GLOBALCONSTANTS DefaultPool_AIC_3P (* Global constants *)
  PACKAGE Uebungen::const::UT::AIC;
  VAR_GLOBAL CONSTANT
    ISO_DESIGNATOR_WIDTH : UINT := 80;
    ISO_DESIGNATOR_HEIGHT : UINT := 80;
    ISO_MASK_SIZE : UINT := 480;
    ISO_VERSION_LABEL : STRING;
    MASK_WIDTH : UINT := 480;
    MASK_HEIGHT : UINT := 480;
    WorkingSet : UINT := 0;
    Macro_M1 : UINT := 1;
    Macro_AIC_1 : UINT := 2;
    Macro_AIC_2 : UINT := 3;
    Macro_AIC_3 : UINT := 4;
    Macro_AIC_4 : UINT := 5;
    DataMask_M1 : UINT := 1000;
    DataMask_AIC1 : UINT := 1001;
    DataMask_AIC2 : UINT := 1002;
    DataMask_AIC3 : UINT := 1003;
    DataMask_AIC4 : UINT := 1004;
    Container_Q : UINT := 3000;
    SoftKeyMask_AIC : UINT := 4000;
    SoftKey_Ausgaenge : UINT := 5000;
    SoftKey_AIC1 : UINT := 5001;
    SoftKey_AIC2 : UINT := 5002;
    SoftKey_AIC3 : UINT := 5003;
    SoftKey_AIC4 : UINT := 5004;
    Button_Q01 : UINT := 6001;
    Button_Q02 : UINT := 6002;
    Button_Q03 : UINT := 6003;
    Button_Q04 : UINT := 6004;
    Button_Q05 : UINT := 6005;
    Button_Q06 : UINT := 6006;
    Button_Q07 : UINT := 6007;
    Button_Q08 : UINT := 6008;
    Button_Q09 : UINT := 6009;
    Button_Q10 : UINT := 6010;
    Button_Q11 : UINT := 6011;
    Button_Q12 : UINT := 6012;
    Button_AIC_I01_CO : UINT := 6013;
    Button_AIC_I01_CS : UINT := 6014;
    Button_AIC_I02_CO : UINT := 6015;
    Button_AIC_I02_CS : UINT := 6016;
    Button_AIC_I03_CO : UINT := 6017;
    Button_AIC_I03_CS : UINT := 6018;
    Button_AIC_I04_CO : UINT := 6019;
    Button_AIC_I04_CS : UINT := 6020;
    Button_AIC_I05_CO : UINT := 6021;
    Button_AIC_I05_CS : UINT := 6022;
    Button_AIC_I06_CO : UINT := 6023;
    Button_AIC_I06_CS : UINT := 6024;
    Button_AIC_I07_CO : UINT := 6025;
    Button_AIC_I07_CS : UINT := 6026;
    Button_AIC_I08_CO : UINT := 6027;
    Button_AIC_I08_CS : UINT := 6028;
    Button_AIC_I01_MID : UINT := 6029;
    Button_AIC_I02_MID : UINT := 6030;
    Button_AIC_I03_MID : UINT := 6031;
    Button_AIC_I04_MID : UINT := 6032;
    Button_AIC_I05_MID : UINT := 6033;
    Button_AIC_I06_MID : UINT := 6034;
    Button_AIC_I07_MID : UINT := 6035;
    Button_AIC_I08_MID : UINT := 6036;
    InputNumber_AIC_I01_ZERO : UINT := 9000;
    InputNumber_AIC_I01_SPAN : UINT := 9001;
    InputNumber_AIC_I02_ZERO : UINT := 9002;
    InputNumber_AIC_I02_SPAN : UINT := 9003;
    InputNumber_AIC_I03_ZERO : UINT := 9004;
    InputNumber_AIC_I03_SPAN : UINT := 9005;
    InputNumber_AIC_I04_ZERO : UINT := 9006;
    InputNumber_AIC_I04_SPAN : UINT := 9007;
    InputNumber_AIC_I05_ZERO : UINT := 9008;
    InputNumber_AIC_I05_SPAN : UINT := 9009;
    InputNumber_AIC_I06_ZERO : UINT := 9010;
    InputNumber_AIC_I06_SPAN : UINT := 9011;
    InputNumber_AIC_I07_ZERO : UINT := 9012;
    InputNumber_AIC_I07_SPAN : UINT := 9013;
    InputNumber_AIC_I08_ZERO : UINT := 9014;
    InputNumber_AIC_I08_SPAN : UINT := 9015;
    InputNumber_AIC_I01_MID : UINT := 9016;
    InputNumber_AIC_I02_MID : UINT := 9017;
    InputNumber_AIC_I03_MID : UINT := 9018;
    InputNumber_AIC_I04_MID : UINT := 9019;
    InputNumber_AIC_I05_MID : UINT := 9020;
    InputNumber_AIC_I06_MID : UINT := 9021;
    InputNumber_AIC_I07_MID : UINT := 9022;
    InputNumber_AIC_I08_MID : UINT := 9023;
    OutputString_WorkingSet_0 : UINT := 11000;
    Label_SoftKey_Ausgaenge : UINT := 11001;
    Label_SoftKey_AIC1 : UINT := 11002;
    Label_SoftKey_AIC2 : UINT := 11003;
    Label_SoftKey_AIC3 : UINT := 11004;
    Label_SoftKey_AIC4 : UINT := 11005;
    Label_AIC_I01 : UINT := 11006;
    Label_AIC_I02 : UINT := 11007;
    Label_AIC_I03 : UINT := 11008;
    Label_AIC_I04 : UINT := 11009;
    Label_AIC_I05 : UINT := 11010;
    Label_AIC_I06 : UINT := 11011;
    Label_AIC_I07 : UINT := 11012;
    Label_AIC_I08 : UINT := 11013;
    Caption_MIN : UINT := 11014;
    Caption_MAX : UINT := 11015;
    Caption_MID : UINT := 11016;
    OutputNumber_c1 : UINT := 12001;
    OutputNumber_c9 : UINT := 12009;
    OutputNumber_c10 : UINT := 12010;
    OutputNumber_c11 : UINT := 12011;
    OutputNumber_c12 : UINT := 12012;
    OutputNumber_c2 : UINT := 12013;
    OutputNumber_c3 : UINT := 12014;
    OutputNumber_c4 : UINT := 12015;
    OutputNumber_c5 : UINT := 12016;
    OutputNumber_c6 : UINT := 12017;
    OutputNumber_c7 : UINT := 12018;
    OutputNumber_c8 : UINT := 12019;
    OutputNumber_Tick : UINT := 12020;
    OutputNumber_AIC_I01_RAW : UINT := 12021;
    OutputNumber_AIC_I01_CAL : UINT := 12022;
    OutputNumber_AIC_I02_RAW : UINT := 12023;
    OutputNumber_AIC_I02_CAL : UINT := 12024;
    OutputNumber_AIC_I03_RAW : UINT := 12025;
    OutputNumber_AIC_I03_CAL : UINT := 12026;
    OutputNumber_AIC_I04_RAW : UINT := 12027;
    OutputNumber_AIC_I04_CAL : UINT := 12028;
    OutputNumber_AIC_I05_RAW : UINT := 12029;
    OutputNumber_AIC_I05_CAL : UINT := 12030;
    OutputNumber_AIC_I06_RAW : UINT := 12031;
    OutputNumber_AIC_I06_CAL : UINT := 12032;
    OutputNumber_AIC_I07_RAW : UINT := 12033;
    OutputNumber_AIC_I07_CAL : UINT := 12034;
    OutputNumber_AIC_I08_RAW : UINT := 12035;
    OutputNumber_AIC_I08_CAL : UINT := 12036;
    OutputNumber_AIC_I01_MINRAW : UINT := 12037;
    OutputNumber_AIC_I01_MIDRAW : UINT := 12038;
    OutputNumber_AIC_I01_MAXRAW : UINT := 12039;
    OutputNumber_AIC_I02_MINRAW : UINT := 12040;
    OutputNumber_AIC_I02_MIDRAW : UINT := 12041;
    OutputNumber_AIC_I02_MAXRAW : UINT := 12042;
    OutputNumber_AIC_I03_MINRAW : UINT := 12043;
    OutputNumber_AIC_I03_MIDRAW : UINT := 12044;
    OutputNumber_AIC_I03_MAXRAW : UINT := 12045;
    OutputNumber_AIC_I04_MINRAW : UINT := 12046;
    OutputNumber_AIC_I04_MIDRAW : UINT := 12047;
    OutputNumber_AIC_I04_MAXRAW : UINT := 12048;
    OutputNumber_AIC_I05_MINRAW : UINT := 12049;
    OutputNumber_AIC_I05_MIDRAW : UINT := 12050;
    OutputNumber_AIC_I05_MAXRAW : UINT := 12051;
    OutputNumber_AIC_I06_MINRAW : UINT := 12052;
    OutputNumber_AIC_I06_MIDRAW : UINT := 12053;
    OutputNumber_AIC_I06_MAXRAW : UINT := 12054;
    OutputNumber_AIC_I07_MINRAW : UINT := 12055;
    OutputNumber_AIC_I07_MIDRAW : UINT := 12056;
    OutputNumber_AIC_I07_MAXRAW : UINT := 12057;
    OutputNumber_AIC_I08_MINRAW : UINT := 12058;
    OutputNumber_AIC_I08_MIDRAW : UINT := 12059;
    OutputNumber_AIC_I08_MAXRAW : UINT := 12060;
    Bargraph_AIC_I01 : UINT := 18000;
    Bargraph_AIC_I02 : UINT := 18001;
    Bargraph_AIC_I03 : UINT := 18002;
    Bargraph_AIC_I04 : UINT := 18003;
    Bargraph_AIC_I05 : UINT := 18004;
    Bargraph_AIC_I06 : UINT := 18005;
    Bargraph_AIC_I07 : UINT := 18006;
    Bargraph_AIC_I08 : UINT := 18007;
    Logos_icon : UINT := 20500;
    NumberVariable_AIC_RAW_I01 : UINT := 21000;
    NumberVariable_AIC_RAW_I02 : UINT := 21001;
    NumberVariable_AIC_RAW_I03 : UINT := 21002;
    NumberVariable_AIC_RAW_I04 : UINT := 21003;
    NumberVariable_AIC_RAW_I05 : UINT := 21004;
    NumberVariable_AIC_RAW_I06 : UINT := 21005;
    NumberVariable_AIC_RAW_I07 : UINT := 21006;
    NumberVariable_AIC_RAW_I08 : UINT := 21007;
    NumberVariable_AIC_CAL_I01 : UINT := 21008;
    NumberVariable_AIC_CAL_I02 : UINT := 21009;
    NumberVariable_AIC_CAL_I03 : UINT := 21010;
    NumberVariable_AIC_CAL_I04 : UINT := 21011;
    NumberVariable_AIC_CAL_I05 : UINT := 21012;
    NumberVariable_AIC_CAL_I06 : UINT := 21013;
    NumberVariable_AIC_CAL_I07 : UINT := 21014;
    NumberVariable_AIC_CAL_I08 : UINT := 21015;
    NumberVariable_AIC_I01_ZERO : UINT := 21016;
    NumberVariable_AIC_I01_SPAN : UINT := 21017;
    NumberVariable_AIC_I02_ZERO : UINT := 21018;
    NumberVariable_AIC_I02_SPAN : UINT := 21019;
    NumberVariable_AIC_I03_ZERO : UINT := 21020;
    NumberVariable_AIC_I03_SPAN : UINT := 21021;
    NumberVariable_AIC_I04_ZERO : UINT := 21022;
    NumberVariable_AIC_I04_SPAN : UINT := 21023;
    NumberVariable_AIC_I05_ZERO : UINT := 21024;
    NumberVariable_AIC_I05_SPAN : UINT := 21025;
    NumberVariable_AIC_I06_ZERO : UINT := 21026;
    NumberVariable_AIC_I06_SPAN : UINT := 21027;
    NumberVariable_AIC_I07_ZERO : UINT := 21028;
    NumberVariable_AIC_I07_SPAN : UINT := 21029;
    NumberVariable_AIC_I08_ZERO : UINT := 21030;
    NumberVariable_AIC_I08_SPAN : UINT := 21031;
    NumberVariable_AIC_I01_MID : UINT := 21032;
    NumberVariable_AIC_I02_MID : UINT := 21033;
    NumberVariable_AIC_I03_MID : UINT := 21034;
    NumberVariable_AIC_I04_MID : UINT := 21035;
    NumberVariable_AIC_I05_MID : UINT := 21036;
    NumberVariable_AIC_I06_MID : UINT := 21037;
    NumberVariable_AIC_I07_MID : UINT := 21038;
    NumberVariable_AIC_I08_MID : UINT := 21039;
    NumberVariable_AIC_I01_MINRAW : UINT := 21040;
    NumberVariable_AIC_I01_MIDRAW : UINT := 21041;
    NumberVariable_AIC_I01_MAXRAW : UINT := 21042;
    NumberVariable_AIC_I02_MINRAW : UINT := 21043;
    NumberVariable_AIC_I02_MIDRAW : UINT := 21044;
    NumberVariable_AIC_I02_MAXRAW : UINT := 21045;
    NumberVariable_AIC_I03_MINRAW : UINT := 21046;
    NumberVariable_AIC_I03_MIDRAW : UINT := 21047;
    NumberVariable_AIC_I03_MAXRAW : UINT := 21048;
    NumberVariable_AIC_I04_MINRAW : UINT := 21049;
    NumberVariable_AIC_I04_MIDRAW : UINT := 21050;
    NumberVariable_AIC_I04_MAXRAW : UINT := 21051;
    NumberVariable_AIC_I05_MINRAW : UINT := 21052;
    NumberVariable_AIC_I05_MIDRAW : UINT := 21053;
    NumberVariable_AIC_I05_MAXRAW : UINT := 21054;
    NumberVariable_AIC_I06_MINRAW : UINT := 21055;
    NumberVariable_AIC_I06_MIDRAW : UINT := 21056;
    NumberVariable_AIC_I06_MAXRAW : UINT := 21057;
    NumberVariable_AIC_I07_MINRAW : UINT := 21058;
    NumberVariable_AIC_I07_MIDRAW : UINT := 21059;
    NumberVariable_AIC_I07_MAXRAW : UINT := 21060;
    NumberVariable_AIC_I08_MINRAW : UINT := 21061;
    NumberVariable_AIC_I08_MIDRAW : UINT := 21062;
    NumberVariable_AIC_I08_MAXRAW : UINT := 21063;
    FontAttributes_6x8 : UINT := 23000;
    FontAttributes_24x32 : UINT := 23001;
    FontAttributes_16x16 : UINT := 23002;
    AuxFunction2_X1 : UINT := 31000;
  END_VAR
END_GLOBALCONSTANTS
